// TIA Portal V18 export
DATA_BLOCK "Aux_Functions_DB"   // DB16
// stored: AutoNumber false, InstanceOfName Aux_Functions, InstanceOfType FB
"Aux_Functions"
   // VAR
   //    PTO_Pulse { S7_SetPoint := 'True'} : TP_TIME;
   //    BUWOpenCLKTOffTime { S7_SetPoint := 'True'} : TP_TIME;
   //    BUWOpenCLKOnTime { S7_SetPoint := 'True'} : TP_TIME;
   //    BUWCloseHoldTOF { S7_SetPoint := 'True'} : TOF_TIME;
   //    MUDoneTP { S7_SetPoint := 'True'} : TP_TIME;
   //    BUWOpPulse { S7_SetPoint := 'True'} : TP_TIME;
   //    ElevCl_TON { S7_SetPoint := 'True'} : TON_TIME;
   //    ElevOpTime_TP { S7_SetPoint := 'True'} : TP_TIME;
   //    MSVOp_TON { S7_SetPoint := 'True'} : TON_TIME;
   //    MPRunning_TOF { S7_SetPoint := 'True'} : TOF_TIME;
   //    MSVCl_TON { S7_SetPoint := 'True'} : TON_TIME;
   //    BUWMainCl_Int { S7_SetPoint := 'True'} : Bool;
   //    TDModeMUTrig : Bool;
   //    TDModeBOTrig { ExternalAccessible := 'False'; ExternalVisible := 'False'; ExternalWritable := 'False'} : Bool;
   //    ElevOpOnTime : Bool;
   //    LinksDisable : Bool;
   //    ElevClDisable : Bool;
   //    MSVClDisable { S7_SetPoint := 'True'} : Bool;
   //    MSVOpDisable { S7_SetPoint := 'True'} : Bool;
   //    ElevOpSwTrig : Bool;
   //    ElevCl_TON_1 { S7_SetPoint := 'True'} : TON_TIME;
   //    ElevCl_TON_5s { S7_SetPoint := 'True'} : TON_TIME;
   // END_VAR
BEGIN
END_DATA_BLOCK
